// TwinCAT 3 PLC project Motion_Library
// Title: MotionControl_Lib
// Company: Chua Siang Poh
// Author: Chua Siang Poh
// ProjectVersion: 2.1.0
// ProgramVersion: 3.1.4020.10
// libraries:
//   Tc2_MC2, * (Beckhoff Automation GmbH)
//   Tc2_Standard, * (Beckhoff Automation GmbH)
//   Tc2_System, * (Beckhoff Automation GmbH)
//   Tc3_Module, * (Beckhoff Automation GmbH)
// project tree:
//   Base Component/Class/ M_ACTUATION.TcPOU, M_ACTUATION_EXT.TcPOU
//   Base Component/Data/ E_ACTUATIONSTATE.TcDUT, S_ACTUATIONDATA.TcDUT
//   Base Component/Interface/ IFC_ACTUATION.TcIO
//   Version/ Global_Version.TcGVL
// real-time tasks:
//   TASK PlcTask: cycle T#10ms, priority 20, ADS port 350

// ---- Base Component/Data/E_ACTUATIONSTATE.TcDUT
{attribute 'qualified_only'}
{attribute 'strict'}
TYPE E_ACTUATIONSTATE :
(
	E_MANUAL_ACTUATION := 0,
	E_PTP_ACTUATION,
	E_PTP_ACTUATION_EXECUTING,
	E_SETPOINT_ACTUATION,
	E_SETPOINT_ACTUATION_ACTIVATED
)UDINT;
END_TYPE

// ---- Base Component/Data/S_ACTUATIONDATA.TcDUT
TYPE S_ACTUATIONDATA :
STRUCT
	NC_INTERFACE 		: AXIS_REF;
	PROBE				: TRIGGER_REF;
	
	CALIBRATE_AT_LIMIT : BOOL := TRUE;
	CALIBRATE_AT_MINUS : BOOL := TRUE;
	
	LIMITS_DISABLED : BOOL;
	LIMITS_INVERTED : BOOL;
	
	HW_HOME_INVERTED: BOOL;
	
	HW_ERR AT %I* 	: UDINT;
	HW_POT AT %I* 	: BOOL;
	HW_NOT AT %I* 	: BOOL;
	HW_HOME AT %I* 	: BOOL;
END_STRUCT
END_TYPE

// ---- Version/Global_Version.TcGVL
{attribute 'TcGenerated'}
// This function has been automatically generated from the project information.
VAR_GLOBAL CONSTANT
	{attribute 'const_non_replaced'}
	{attribute 'linkalways'}
	stLibVersion_MotionControl_Lib : ST_LibVersion := (iMajor := 2, iMinor := 1, iBuild := 0, iRevision := 0, sVersion := '2.1.0');
END_VAR

// ---- Base Component/Interface/IFC_ACTUATION.TcIO
INTERFACE IFC_ACTUATION

PROPERTY ACCELERATION : LREAL
GET
END_GET
SET
END_SET
END_PROPERTY

METHOD ACTIVATE_EXTERNAL_SETPOINT : DINT
VAR_INPUT
END_VAR
END_METHOD

METHOD ACTIVATE_TOUCHPROBE : DINT
VAR_INPUT
END_VAR
END_METHOD

PROPERTY AT_NEGATIVE_LIMIT : BOOL
GET
END_GET
END_PROPERTY

PROPERTY AT_POSITIVE_LIMIT : BOOL
GET
END_GET
END_PROPERTY

PROPERTY AXIS_ERROR : BOOL
GET
END_GET
END_PROPERTY

PROPERTY AXIS_ERROR_ID : UDINT
GET
END_GET
END_PROPERTY

PROPERTY CALIBRATE_AT_LIMIT : BOOL
GET
END_GET
SET
END_SET
END_PROPERTY

PROPERTY CALIBRATE_TO_NEGATIVE : BOOL
GET
END_GET
SET
END_SET
END_PROPERTY

METHOD DEACTIVATE_EXTERNAL_SETPOINT : DINT
VAR_INPUT
END_VAR
END_METHOD

METHOD DEACTIVATE_TOUCHPROBE : DINT
VAR_INPUT
END_VAR
END_METHOD

PROPERTY DECELERATION : LREAL
GET
END_GET
SET
END_SET
END_PROPERTY

PROPERTY DISABLE_LIMITS : BOOL
GET
END_GET
SET
END_SET
END_PROPERTY

PROPERTY ENABLE : BOOL
GET
END_GET
SET
END_SET
END_PROPERTY

METHOD HALT : DINT
VAR_INPUT
END_VAR
END_METHOD

PROPERTY HARDWARE_ERROR_CODE : UDINT
GET
END_GET
END_PROPERTY

PROPERTY HAS_JOB : BOOL
GET
END_GET
END_PROPERTY

METHOD HOME : DINT
VAR_INPUT
END_VAR
END_METHOD

METHOD HOME_FORCED : DINT
VAR_INPUT
END_VAR
END_METHOD

PROPERTY ID : UDINT
GET
END_GET
END_PROPERTY

PROPERTY INVERT_CALIBRATION_SIGNAL : BOOL
GET
END_GET
SET
END_SET
END_PROPERTY

PROPERTY INVERT_LIMITS : BOOL
GET
END_GET
SET
END_SET
END_PROPERTY

PROPERTY IS_MOVING : BOOL
GET
END_GET
END_PROPERTY

PROPERTY JERK : LREAL
GET
END_GET
SET
END_SET
END_PROPERTY

PROPERTY JOG_BACKWARD : BOOL
SET
END_SET
END_PROPERTY

PROPERTY JOG_FORWARD : BOOL
SET
END_SET
END_PROPERTY

PROPERTY JOG_VELOCITY : LREAL
GET
END_GET
SET
END_SET
END_PROPERTY

PROPERTY MODE : E_ACTUATIONSTATE
GET
END_GET
SET
END_SET
END_PROPERTY

METHOD MOVE_ALONG : LREAL
VAR_INPUT
	VELOCITY	: LREAL;
	FORWARD 	: BOOL;
END_VAR
END_METHOD

METHOD MOVE_BY : DINT
VAR_INPUT
	DISTANCE : LREAL;
	VELOCITY : LREAL;
END_VAR
END_METHOD

METHOD MOVE_TO : DINT
VAR_INPUT
	POSITION : LREAL;
	VELOCITY : LREAL;
END_VAR
END_METHOD

PROPERTY OVERRIDE : LREAL
GET
END_GET
SET
END_SET
END_PROPERTY

PROPERTY POSITION : LREAL
GET
END_GET
END_PROPERTY

METHOD RESET : DINT
VAR_INPUT
END_VAR
END_METHOD

PROPERTY SET_DIRECTION : DINT
SET
END_SET
END_PROPERTY

PROPERTY SET_POSITION : LREAL
SET
END_SET
END_PROPERTY

PROPERTY SET_VELOCITY : LREAL
SET
END_SET
END_PROPERTY

PROPERTY VELOCITY : LREAL
GET
END_GET
END_PROPERTY

END_INTERFACE

// ---- Base Component/Class/M_ACTUATION.TcPOU
FUNCTION_BLOCK M_ACTUATION IMPLEMENTS IFC_ACTUATION
VAR_INPUT
END_VAR
VAR_OUTPUT
	STATE : E_ACTUATIONSTATE;
END_VAR
VAR	
	AXIS : S_ACTUATIONDATA;
	
	MOTION_ACCELERATION : LREAL := 0;
	MOTION_DECELERATION : LREAL := 0;
	MOTION_JERK 		: LREAL := 0;
	
	_PROBEPOSITION	: LREAL;
	_PROBEDATA		: MC_TouchProbeRecordedData;
	_FBTPROBE		: MC_TOUCHPROBE;
	_FBTPROBE_ABORT	: MC_ABORTTRIGGER;
	
	MANUAL_FORWARD 	: BOOL;
	MANUAL_BACKWARD : BOOL;
	_FBPOWER 		: MC_POWER;
	_FBRESET		: MC_RESET;
	_FBHALT			: MC_HALT;
	_FBHOME			: MC_HOME;
	_FBJOG			: MC_JOG;
	_FBMOVEABS		: MC_MOVEABSOLUTE;
	_FBMOVEREL		: MC_MOVERELATIVE;
	_FBMOVEVEL		: MC_MOVEVELOCITY;
	
	SETPOINT_POSITION 		: LREAL;
	SETPOINT_VELOCITY 		: LREAL;
	SETPOINT_DIRECTION		: DINT;
	
	_FBEXTEN		: MC_ExtSetPointGenEnable;
	_FBEXTDN		: MC_ExtSetPointGenDisable;
	//_FBEXTFEED		: MC_ExtSetPointGenFeed;
END_VAR

_FBPOWER.Enable_Positive := (NOT(AXIS.HW_POT XOR AXIS.LIMITS_INVERTED)) OR DISABLE_LIMITS;
_FBPOWER.Enable_Negative := (NOT(AXIS.HW_NOT XOR AXIS.LIMITS_INVERTED)) OR DISABLE_LIMITS;
_FBPOWER(Axis:= AXIS.NC_INTERFACE);

CASE STATE OF 
	E_ACTUATIONSTATE.E_MANUAL_ACTUATION:
		_FBJOG(
			Axis:= AXIS.NC_INTERFACE, 
			JogForward:= MANUAL_FORWARD AND ENABLE, 
			JogBackwards:= MANUAL_BACKWARD AND ENABLE, 
			Mode:= MC_JOGMODE_CONTINOUS, 
			Velocity:= , 
			Acceleration:= ACCELERATION, 
			Deceleration:= DECELERATION, 
			Jerk:= JERK ); 
	ELSE
		_FBJOG(
			Axis:= AXIS.NC_INTERFACE, 
			JogForward:= FALSE, 
			JogBackwards:= FALSE );
END_CASE
CASE STATE OF 
	E_ACTUATIONSTATE.E_SETPOINT_ACTUATION_ACTIVATED:
		AXIS.NC_INTERFACE.PlcToNc.ExtSetPos := SETPOINT_POSITION;
		AXIS.NC_INTERFACE.PlcToNc.ExtSetVelo := SETPOINT_VELOCITY;
		AXIS.NC_INTERFACE.PlcToNc.ExtSetDirection := SETPOINT_DIRECTION;
	ELSE
		;
END_CASE

PROPERTY ACCELERATION : LREAL
GET
ACCELERATION := MOTION_ACCELERATION;
END_GET
SET
MOTION_ACCELERATION := ABS(ACCELERATION);
END_SET
END_PROPERTY

METHOD ACTIVATE_EXTERNAL_SETPOINT : DINT
VAR_INPUT
END_VAR
CASE STATE OF 
	E_ACTUATIONSTATE.E_SETPOINT_ACTUATION:
		_FBEXTEN(
			Axis:= AXIS.NC_INTERFACE, 
			Execute:= TRUE, 
			Position:= , 
			PositionType:= POSITIONTYPE_ABSOLUTE );
		IF _FBEXTEN.Error THEN
			_FBEXTEN(
				Axis:= AXIS.NC_INTERFACE, 
				Execute:= FALSE );
			STATE := E_ACTUATIONSTATE.E_SETPOINT_ACTUATION;
			ACTIVATE_EXTERNAL_SETPOINT := 1;
			RETURN;
		ELSIF _FBEXTEN.Done THEN
			_FBEXTEN(
				Axis:= AXIS.NC_INTERFACE, 
				Execute:= FALSE );
			STATE := E_ACTUATIONSTATE.E_SETPOINT_ACTUATION_ACTIVATED;
			ACTIVATE_EXTERNAL_SETPOINT := -1;
			RETURN;
		ELSE
			STATE := E_ACTUATIONSTATE.E_SETPOINT_ACTUATION;
			ACTIVATE_EXTERNAL_SETPOINT := 0;
			RETURN;
		END_IF
	ELSE 
		ACTIVATE_EXTERNAL_SETPOINT := 99;
		RETURN;
END_CASE
END_METHOD

METHOD ACTIVATE_TOUCHPROBE : DINT
VAR_INPUT
END_VAR
_FBTPROBE(
	Axis:= AXIS.NC_INTERFACE, 
	TriggerInput:= AXIS.PROBE, 
	Execute:= TRUE, 
	WindowOnly:= FALSE, 
	FirstPosition:= , 
	LastPosition:= , 
	Done=> , 
	Busy=> , 
	CommandAborted=> , 
	Error=> , 
	ErrorID=> , 
	RecordedPosition=> , 
	RecordedData=> );
IF _FBTPROBE.Error OR _FBTPROBE.CommandAborted THEN
	_FBTPROBE(
		Axis:= AXIS.NC_INTERFACE, 
		TriggerInput:= AXIS.PROBE, 
		Execute:= FALSE );
	ACTIVATE_TOUCHPROBE := 1;
	RETURN;
ELSIF _FBTPROBE.Done THEN
	_FBTPROBE(
		Axis:= AXIS.NC_INTERFACE, 
		TriggerInput:= AXIS.PROBE, 
		Execute:= FALSE );
	_PROBEDATA := _FBTPROBE.RecordedData;
	_PROBEPOSITION := _FBTPROBE.RecordedPosition;
	ACTIVATE_TOUCHPROBE := -1;
	RETURN;
ELSE
	_FBTPROBE(
		Axis:= AXIS.NC_INTERFACE, 
		TriggerInput:= AXIS.PROBE, 
		Execute:= FALSE );
	ACTIVATE_TOUCHPROBE := 0;
	RETURN;
END_IF
END_METHOD

PROPERTY AT_NEGATIVE_LIMIT : BOOL
GET
AT_NEGATIVE_LIMIT := AXIS.HW_NOT;
END_GET
END_PROPERTY

PROPERTY AT_POSITIVE_LIMIT : BOOL
GET
AT_POSITIVE_LIMIT := AXIS.HW_POT;
END_GET
END_PROPERTY

PROPERTY AXIS_ERROR : BOOL
GET
AXIS.NC_INTERFACE.ReadStatus();
AXIS_ERROR := AXIS.NC_INTERFACE.Status.Error;
END_GET
END_PROPERTY

PROPERTY AXIS_ERROR_ID : UDINT
GET
AXIS_ERROR_ID := AXIS.NC_INTERFACE.NcToPlc.ErrorCode;
END_GET
END_PROPERTY

PROPERTY CALIBRATE_AT_LIMIT : BOOL
GET
CALIBRATE_AT_LIMIT := AXIS.CALIBRATE_AT_LIMIT;
END_GET
SET
AXIS.CALIBRATE_AT_LIMIT := CALIBRATE_AT_LIMIT;
END_SET
END_PROPERTY

PROPERTY CALIBRATE_TO_NEGATIVE : BOOL
GET
CALIBRATE_TO_NEGATIVE := AXIS.CALIBRATE_AT_MINUS;
END_GET
SET
AXIS.CALIBRATE_AT_MINUS := CALIBRATE_TO_NEGATIVE;
END_SET
END_PROPERTY

METHOD DEACTIVATE_EXTERNAL_SETPOINT : DINT
VAR_INPUT
END_VAR
CASE STATE OF 
	E_ACTUATIONSTATE.E_SETPOINT_ACTUATION_ACTIVATED:
		_FBEXTDN(
			Axis:= AXIS.NC_INTERFACE, 
			Execute:= TRUE );
		IF _FBEXTDN.Error THEN
			_FBEXTDN(
				Axis:= AXIS.NC_INTERFACE, 
				Execute:= FALSE );
			STATE := E_ACTUATIONSTATE.E_SETPOINT_ACTUATION_ACTIVATED;
			DEACTIVATE_EXTERNAL_SETPOINT := 1;
			RETURN;
		ELSIF _FBEXTDN.Done THEN
			_FBEXTDN(
				Axis:= AXIS.NC_INTERFACE, 
				Execute:= FALSE );
			STATE := E_ACTUATIONSTATE.E_SETPOINT_ACTUATION;
			DEACTIVATE_EXTERNAL_SETPOINT := -1;
			RETURN;
		ELSE
			STATE := E_ACTUATIONSTATE.E_SETPOINT_ACTUATION_ACTIVATED;
			DEACTIVATE_EXTERNAL_SETPOINT := 0;
			RETURN;
		END_IF
	ELSE 
		DEACTIVATE_EXTERNAL_SETPOINT := 99;
		RETURN;
END_CASE
END_METHOD

METHOD DEACTIVATE_TOUCHPROBE : DINT
VAR_INPUT
END_VAR
_FBTPROBE_ABORT(
	Axis:= AXIS.NC_INTERFACE, 
	TriggerInput:= AXIS.PROBE, 
	Execute:= TRUE );
IF _FBTPROBE_ABORT.Error THEN
	_FBTPROBE_ABORT(
		Axis:= AXIS.NC_INTERFACE, 
		TriggerInput:= AXIS.PROBE, 
		Execute:= FALSE );
	DEACTIVATE_TOUCHPROBE := 1;
	RETURN;
ELSIF _FBTPROBE_ABORT.DONE THEN
	_FBTPROBE_ABORT(
		Axis:= AXIS.NC_INTERFACE, 
		TriggerInput:= AXIS.PROBE, 
		Execute:= FALSE );
	DEACTIVATE_TOUCHPROBE := -1;
	RETURN; 
ELSE
	DEACTIVATE_TOUCHPROBE := 0;
	RETURN; 
END_IF
END_METHOD

PROPERTY DECELERATION : LREAL
GET
DECELERATION := MOTION_DECELERATION;
END_GET
SET
MOTION_DECELERATION := ABS(DECELERATION);
END_SET
END_PROPERTY

PROPERTY DISABLE_LIMITS : BOOL
GET
DISABLE_LIMITS := AXIS.LIMITS_DISABLED;
END_GET
SET
AXIS.LIMITS_DISABLED := DISABLE_LIMITS;
END_SET
END_PROPERTY

PROPERTY ENABLE : BOOL
GET
ENABLE := _FBPOWER.Status;
END_GET
SET
_FBPOWER.Enable := ENABLE;
END_SET
END_PROPERTY

METHOD HALT : DINT
VAR_INPUT
END_VAR
THIS^.JOG_FORWARD := FALSE;
THIS^.JOG_BACKWARD := FALSE;

_FBHALT(
	Axis:= AXIS.NC_INTERFACE, 
	Execute:= TRUE, 
	Deceleration:= DECELERATION, 
	Jerk:= JERK );
IF _FBHALT.Error THEN
	_FBHALT(
		Axis:= AXIS.NC_INTERFACE, 
		Execute:= FALSE );
	HALT := 1;
	RETURN;
ELSIF _FBHALT.CommandAborted THEN
	_FBHALT(
		Axis:= AXIS.NC_INTERFACE, 
		Execute:= FALSE );
	HALT := 2;
	RETURN;
ELSIF _FBHALT.Done THEN
	_FBHALT(
		Axis:= AXIS.NC_INTERFACE, 
		Execute:= FALSE );
	HALT := -1;
	RETURN;
ELSE
	HALT := 0;
	RETURN;
END_IF
END_METHOD

PROPERTY HARDWARE_ERROR_CODE : UDINT
GET
HARDWARE_ERROR_CODE := AXIS.HW_ERR;
END_GET
END_PROPERTY

PROPERTY HAS_JOB : BOOL
GET
AXIS.NC_INTERFACE.ReadStatus();
HAS_JOB := AXIS.NC_INTERFACE.Status.HasJob;
END_GET
END_PROPERTY

METHOD HOME : DINT
VAR_INPUT
END_VAR
CASE STATE OF 
	E_ACTUATIONSTATE.E_PTP_ACTUATION, E_ACTUATIONSTATE.E_PTP_ACTUATION_EXECUTING:
		DISABLE_LIMITS := TRUE;
		IF AXIS.CALIBRATE_AT_LIMIT THEN
			IF AXIS.CALIBRATE_AT_MINUS THEN
				_FBHOME.bCalibrationCam := AXIS.HW_NOT XOR AXIS.LIMITS_INVERTED;
			ELSE
				_FBHOME.bCalibrationCam := AXIS.HW_POT XOR AXIS.LIMITS_INVERTED;
			END_IF
		ELSE
			_FBHOME.bCalibrationCam := AXIS.HW_HOME XOR AXIS.HW_HOME_INVERTED;
		END_IF
		_FBHOME(
			Axis:= AXIS.NC_INTERFACE, 
			Execute:= TRUE, 
			Position:= , 
			HomingMode:= MC_DEFAULTHOMING, 
			bCalibrationCam:= );
		IF _FBHOME.Error THEN
			_FBHOME(
				Axis:= AXIS.NC_INTERFACE, 
				Execute:= FALSE);
			STATE := E_ACTUATIONSTATE.E_PTP_ACTUATION;
			DISABLE_LIMITS := FALSE;
			HOME := 1;
			RETURN;
		ELSIF _FBHOME.CommandAborted THEN
			_FBHOME(
				Axis:= AXIS.NC_INTERFACE, 
				Execute:= FALSE);
			STATE := E_ACTUATIONSTATE.E_PTP_ACTUATION;
			DISABLE_LIMITS := FALSE;
			HOME := 2;
			RETURN;
		ELSIF _FBHOME.Done THEN
			_FBHOME(
				Axis:= AXIS.NC_INTERFACE, 
				Execute:= FALSE);
			STATE := E_ACTUATIONSTATE.E_PTP_ACTUATION;
			DISABLE_LIMITS := FALSE;
			HOME := -1;
			RETURN;
		ELSE
			STATE := E_ACTUATIONSTATE.E_PTP_ACTUATION_EXECUTING;
			HOME := 0;
			RETURN;
		END_IF
END_CASE
END_METHOD

METHOD HOME_FORCED : DINT
VAR_INPUT
END_VAR
CASE STATE OF 
	E_ACTUATIONSTATE.E_PTP_ACTUATION, E_ACTUATIONSTATE.E_PTP_ACTUATION_EXECUTING:
		_FBHOME(
			Axis:= AXIS.NC_INTERFACE, 
			Execute:= TRUE, 
			Position:= , 
			HomingMode:= MC_DIRECT, 
			bCalibrationCam:= );
		IF _FBHOME.Error THEN
			_FBHOME(
				Axis:= AXIS.NC_INTERFACE, 
				Execute:= FALSE);
			STATE := E_ACTUATIONSTATE.E_PTP_ACTUATION;
			HOME_FORCED := 1;
			RETURN;
		ELSIF _FBHOME.CommandAborted THEN
			_FBHOME(
				Axis:= AXIS.NC_INTERFACE, 
				Execute:= FALSE);
			STATE := E_ACTUATIONSTATE.E_PTP_ACTUATION;
			HOME_FORCED := 2;
			RETURN;
		ELSIF _FBHOME.Done THEN
			_FBHOME(
				Axis:= AXIS.NC_INTERFACE, 
				Execute:= FALSE);
			STATE := E_ACTUATIONSTATE.E_PTP_ACTUATION;
			HOME_FORCED := -1;
			RETURN;
		ELSE
			STATE := E_ACTUATIONSTATE.E_PTP_ACTUATION_EXECUTING;
			HOME_FORCED := 0;
			RETURN;
		END_IF
END_CASE
END_METHOD

PROPERTY ID : UDINT
GET
ID := AXIS.NC_INTERFACE.NcToPlc.AxisId;
END_GET
END_PROPERTY

PROPERTY INVERT_CALIBRATION_SIGNAL : BOOL
GET
INVERT_CALIBRATION_SIGNAL := AXIS.HW_HOME_INVERTED;
END_GET
SET
AXIS.HW_HOME_INVERTED := INVERT_CALIBRATION_SIGNAL;
END_SET
END_PROPERTY

PROPERTY INVERT_LIMITS : BOOL
GET
INVERT_LIMITS := AXIS.LIMITS_INVERTED;
END_GET
SET
AXIS.LIMITS_INVERTED := INVERT_LIMITS;
END_SET
END_PROPERTY

PROPERTY IS_MOVING : BOOL
GET
AXIS.NC_INTERFACE.ReadStatus();
IS_MOVING := AXIS.NC_INTERFACE.Status.Moving;
END_GET
END_PROPERTY

PROPERTY JERK : LREAL
GET
JERK := MOTION_JERK;
END_GET
SET
MOTION_JERK := ABS(JERK);
END_SET
END_PROPERTY

PROPERTY JOG_BACKWARD : BOOL
SET
MANUAL_BACKWARD := JOG_BACKWARD;
END_SET
END_PROPERTY

PROPERTY JOG_FORWARD : BOOL
SET
MANUAL_FORWARD := JOG_FORWARD;
END_SET
END_PROPERTY

PROPERTY JOG_VELOCITY : LREAL
GET
JOG_VELOCITY := _FBJOG.Velocity;
END_GET
SET
IF JOG_VELOCITY > 0.0 THEN
	_FBJOG.Velocity := JOG_VELOCITY;
END_IF
END_SET
END_PROPERTY

PROPERTY MODE : E_ACTUATIONSTATE
GET
MODE := STATE;
END_GET
SET
CASE MODE OF
E_ACTUATIONSTATE.E_MANUAL_ACTUATION:
	CASE STATE OF 
		E_ACTUATIONSTATE.E_PTP_ACTUATION, E_ACTUATIONSTATE.E_SETPOINT_ACTUATION:
			STATE := MODE;
	END_CASE
E_ACTUATIONSTATE.E_PTP_ACTUATION:
	CASE STATE OF 
		E_ACTUATIONSTATE.E_MANUAL_ACTUATION, E_ACTUATIONSTATE.E_SETPOINT_ACTUATION:
			STATE := MODE;
	END_CASE
E_ACTUATIONSTATE.E_SETPOINT_ACTUATION:
	CASE STATE OF 
		E_ACTUATIONSTATE.E_MANUAL_ACTUATION, E_ACTUATIONSTATE.E_PTP_ACTUATION:
			STATE := MODE;
	END_CASE
END_CASE
END_SET
END_PROPERTY

METHOD MOVE_ALONG : LREAL
VAR_INPUT
	VELOCITY	: LREAL;
	FORWARD 	: BOOL;
END_VAR
CASE STATE OF 
	E_ACTUATIONSTATE.E_PTP_ACTUATION, E_ACTUATIONSTATE.E_PTP_ACTUATION_EXECUTING:
		IF FORWARD THEN
			_FBMOVEVEL.Direction := 1;
		ELSE
			_FBMOVEVEL.Direction := 3;
		END_IF
		_FBMOVEVEL(
			Axis:= AXIS.NC_INTERFACE, 
			Execute:= TRUE, 
			Velocity:= VELOCITY, 
			Acceleration:= ACCELERATION, 
			Deceleration:= DECELERATION, 
			Jerk:= JERK );
		IF _FBMOVEVEL.Error THEN
			_FBMOVEVEL(
				Axis:= AXIS.NC_INTERFACE, 
				Execute:= FALSE);
			STATE := E_ACTUATIONSTATE.E_PTP_ACTUATION;
			MOVE_ALONG := 1;
			RETURN;
		ELSIF _FBMOVEVEL.CommandAborted THEN
			_FBMOVEVEL(
				Axis:= AXIS.NC_INTERFACE, 
				Execute:= FALSE);
			STATE := E_ACTUATIONSTATE.E_PTP_ACTUATION;
			MOVE_ALONG := 2;
			RETURN;
		ELSIF _FBMOVEVEL.InVelocity THEN
			_FBMOVEVEL(
				Axis:= AXIS.NC_INTERFACE, 
				Execute:= FALSE);
			STATE := E_ACTUATIONSTATE.E_PTP_ACTUATION;
			MOVE_ALONG := -1;
			RETURN;
		ELSE
			STATE := E_ACTUATIONSTATE.E_PTP_ACTUATION_EXECUTING;
			MOVE_ALONG := 0;
			RETURN;
		END_IF
	ELSE
		MOVE_ALONG := 99;
		RETURN;
END_CASE
END_METHOD

METHOD MOVE_BY : DINT
VAR_INPUT
	DISTANCE : LREAL;
	VELOCITY : LREAL;
END_VAR
CASE STATE OF 
	E_ACTUATIONSTATE.E_PTP_ACTUATION, E_ACTUATIONSTATE.E_PTP_ACTUATION_EXECUTING:
		_FBMOVEREL(
			Axis:= AXIS.NC_INTERFACE, 
			Execute:= TRUE, 
			Distance:= DISTANCE, 
			Velocity:= VELOCITY, 
			Acceleration:= ACCELERATION, 
			Deceleration:= DECELERATION, 
			Jerk:= JERK );
		IF _FBMOVEREL.Error THEN
			_FBMOVEREL(
				Axis:= AXIS.NC_INTERFACE, 
				Execute:= FALSE );
			STATE := E_ACTUATIONSTATE.E_PTP_ACTUATION;
			MOVE_BY := 1;
			RETURN;
		ELSIF _FBMOVEREL.CommandAborted THEN
			_FBMOVEREL(
				Axis:= AXIS.NC_INTERFACE, 
				Execute:= FALSE );
			STATE := E_ACTUATIONSTATE.E_PTP_ACTUATION;
			MOVE_BY := 2;
			RETURN;
		ELSIF _FBMOVEREL.Done THEN
			_FBMOVEREL(
				Axis:= AXIS.NC_INTERFACE, 
				Execute:= FALSE );
			STATE := E_ACTUATIONSTATE.E_PTP_ACTUATION;
			MOVE_BY := -1;
			RETURN;
		ELSE
			STATE := E_ACTUATIONSTATE.E_PTP_ACTUATION_EXECUTING;
			MOVE_BY := 0;
			RETURN;
		END_IF
	ELSE
		MOVE_BY := 99;
		RETURN;
END_CASE
END_METHOD

METHOD MOVE_TO : DINT
VAR_INPUT
	POSITION : LREAL;
	VELOCITY : LREAL;
END_VAR
CASE STATE OF 
	E_ACTUATIONSTATE.E_PTP_ACTUATION, E_ACTUATIONSTATE.E_PTP_ACTUATION_EXECUTING:
		_FBMOVEABS(
			Axis:= AXIS.NC_INTERFACE, 
			Execute:= TRUE, 
			Position:= POSITION, 
			Velocity:= VELOCITY, 
			Acceleration:= ACCELERATION, 
			Deceleration:= DECELERATION, 
			Jerk:= JERK );
		IF _FBMOVEABS.Error THEN
			_FBMOVEABS(
				Axis:= AXIS.NC_INTERFACE, 
				Execute:= FALSE );
			STATE := E_ACTUATIONSTATE.E_PTP_ACTUATION;
			MOVE_TO := 1;
			RETURN;
		ELSIF _FBMOVEABS.CommandAborted THEN
			_FBMOVEABS(
				Axis:= AXIS.NC_INTERFACE, 
				Execute:= FALSE );
			STATE := E_ACTUATIONSTATE.E_PTP_ACTUATION;
			MOVE_TO := 2;
			RETURN;
		ELSIF _FBMOVEABS.Done THEN
			_FBMOVEABS(
				Axis:= AXIS.NC_INTERFACE, 
				Execute:= FALSE );
			STATE := E_ACTUATIONSTATE.E_PTP_ACTUATION;
			MOVE_TO := -1;
			RETURN;
		ELSE
			STATE := E_ACTUATIONSTATE.E_PTP_ACTUATION_EXECUTING;
			MOVE_TO := 0;
			RETURN;
		END_IF
	ELSE
		MOVE_TO := 99;
		RETURN;
END_CASE
END_METHOD

PROPERTY OVERRIDE : LREAL
GET
Override := _FBPOWER.Override;
END_GET
SET
IF OVERRIDE > 100.0 THEN
	_FBPOWER.Override := 100;
ELSIF OVERRIDE < 0.0 THEN 
	_FBPOWER.Override := 0.0;
ELSE
	_FBPOWER.Override := OVERRIDE;
END_IF
END_SET
END_PROPERTY

PROPERTY POSITION : LREAL
GET
POSITION := AXIS.NC_INTERFACE.NcToPlc.ActPos;
END_GET
END_PROPERTY

METHOD RESET : DINT
VAR_INPUT
END_VAR
_FBRESET(
	Axis:= AXIS.NC_INTERFACE, 
	Execute:= TRUE );
IF _FBRESET.Error THEN
	_FBRESET(
		Axis:= AXIS.NC_INTERFACE, 
		Execute:= FALSE );
	RESET := 1;
	RETURN;
ELSIF _FBRESET.Done THEN
	_FBRESET(
		Axis:= AXIS.NC_INTERFACE, 
		Execute:= FALSE );
	RESET := -1;
	RETURN;
ELSE 
	RESET := 0;
	RETURN;
END_IF
END_METHOD

PROPERTY SET_DIRECTION : DINT
SET
IF SET_DIRECTION >= 1 THEN
	SETPOINT_DIRECTION := 1;
ELSIF SET_DIRECTION <= -1 THEN
	SETPOINT_DIRECTION := -1;
ELSE
	SETPOINT_DIRECTION := 0;
END_IF
END_SET
END_PROPERTY

PROPERTY SET_POSITION : LREAL
SET
SETPOINT_POSITION := SET_POSITION;
END_SET
END_PROPERTY

PROPERTY SET_VELOCITY : LREAL
SET
SETPOINT_VELOCITY := SET_VELOCITY;
END_SET
END_PROPERTY

PROPERTY VELOCITY : LREAL
GET
VELOCITY := AXIS.NC_INTERFACE.NcToPlc.ActVelo;
END_GET
END_PROPERTY

END_FUNCTION_BLOCK

// ---- Base Component/Class/M_ACTUATION_EXT.TcPOU
FUNCTION_BLOCK M_ACTUATION_EXT EXTENDS M_ACTUATION
VAR_INPUT
END_VAR
VAR_OUTPUT
END_VAR
VAR
END_VAR

METHOD HOME_HARDSTOP : DINT
VAR_INPUT
	TOLERANCE : LREAL := 5.0;
END_VAR
CASE STATE OF 
	E_ACTUATIONSTATE.E_PTP_ACTUATION, E_ACTUATIONSTATE.E_PTP_ACTUATION_EXECUTING:
		DISABLE_LIMITS := TRUE;
		_FBHOME.bCalibrationCam := LAG_ERROR > TOLERANCE;
		_FBHOME(
			Axis:= AXIS.NC_INTERFACE, 
			Execute:= TRUE, 
			Position:= , 
			HomingMode:= MC_DEFAULTHOMING, 
			bCalibrationCam:= );
		IF _FBHOME.Error THEN
			_FBHOME(
				Axis:= AXIS.NC_INTERFACE, 
				Execute:= FALSE);
			STATE := E_ACTUATIONSTATE.E_PTP_ACTUATION;
			DISABLE_LIMITS := FALSE;
			HOME := 1;
			RETURN;
		ELSIF _FBHOME.CommandAborted THEN
			_FBHOME(
				Axis:= AXIS.NC_INTERFACE, 
				Execute:= FALSE);
			STATE := E_ACTUATIONSTATE.E_PTP_ACTUATION;
			DISABLE_LIMITS := FALSE;
			HOME := 2;
			RETURN;
		ELSIF _FBHOME.Done THEN
			_FBHOME(
				Axis:= AXIS.NC_INTERFACE, 
				Execute:= FALSE);
			STATE := E_ACTUATIONSTATE.E_PTP_ACTUATION;
			DISABLE_LIMITS := FALSE;
			HOME := -1;
			RETURN;
		ELSE
			STATE := E_ACTUATIONSTATE.E_PTP_ACTUATION_EXECUTING;
			HOME := 0;
			RETURN;
		END_IF
END_CASE
END_METHOD

PROPERTY LAG_ERROR : LREAL
GET
LAG_ERROR := AXIS.NC_INTERFACE.NcToPlc.PosDiff;
END_GET
END_PROPERTY

END_FUNCTION_BLOCK
